TYPE ConveyorConfiguration :
STRUCT
	iNumSensor : DINT;
	iNumRamp : DINT;
	iNumPusher : DINT;
END_STRUCT
END_TYPE

(* stored: Version 1.1.0.1, ProductVersion 3.1.4024.9
   DUT ConveyorConfiguration: Id {4e5f7f49-9963-4557-95cd-0ab3f3b8ec00} *)
